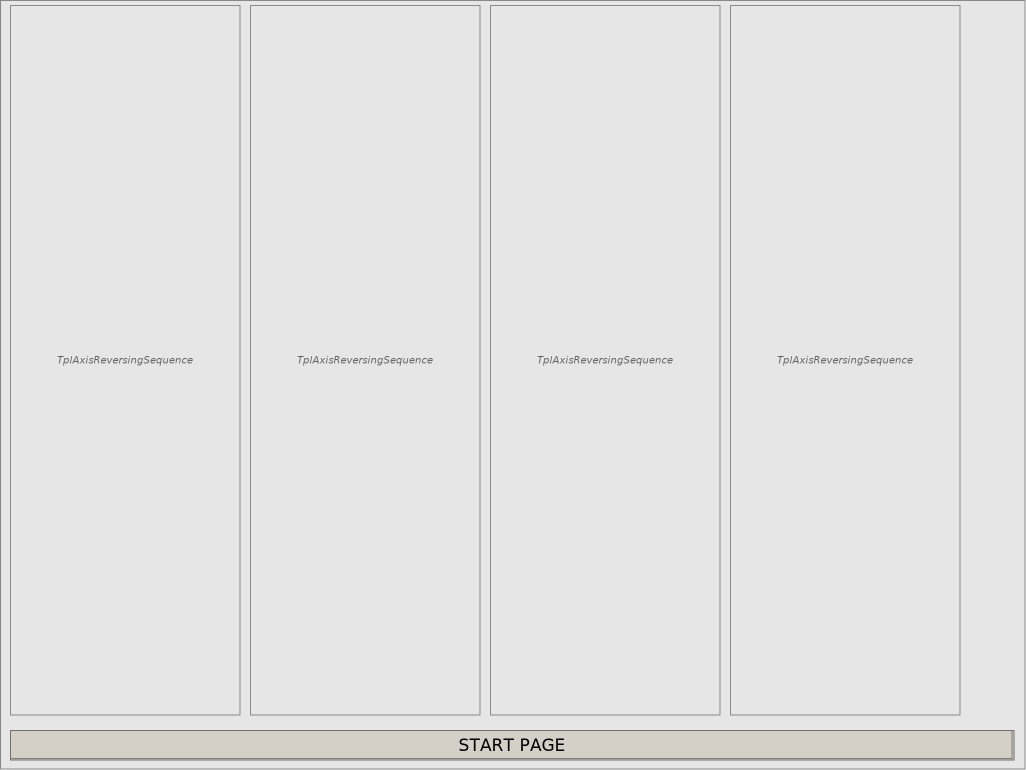
VISUALIZATION HmiAxisReversingSequence  // 1026x770
    Rectangle (0,0 1024x768)
    Button (10,730 1004x30), "START PAGE"
        OnMouseClick: change screen: HmiStartPage
    Frame (10,5 230x710)
        shows TplAxisReversingSequence(sAxisDescription := Axis1.sAxisDescription, fAbsolutePositon := stAxis1.NcToPlc.ActPos, fModuloPositon := stAxis1.NcToPlc.ModuloActPos, bError := Axis1.bAxisErr, nErrorId := Axis1.nAxisErrId, bReset := Axis1.bReset, bPowerStatus := Axis1.fbAxis.bPowerStatus, bReferenceCam := bStepperReferenceCam, bRevSeqStart := Axis1.bRevSeqStart, bRevSeqStop := Axis1.fbAxis.bRevSeqStop, fRevSeqTargetPos1 := Axis1.fbAxis.fRevSeqTargetPos1, fRevSeqTargetVelo1 := Axis1.fbAxis.fRevSeqTargetVelo1, fRevSeqTargetPos2 := Axis1.fbAxis.fRevSeqTargetPos2, fRevSeqTargetVelo2 := Axis1.fbAxis.fRevSeqTargetVelo2, nRevSeqIdleTime := Axis1.fbAxis.nRevSeqIdleTime, bRevSeqDone := Axis1.fbAxis.bRevSeqDone, bRevSeqBusy := Axis1.fbAxis.bRevSeqBusy)
    Frame (250,5 230x710)
        shows TplAxisReversingSequence(sAxisDescription := Axis2.sAxisDescription, fAbsolutePositon := stAxis2.NcToPlc.ActPos, fModuloPositon := stAxis2.NcToPlc.ModuloActPos, bError := Axis2.bAxisErr, nErrorId := Axis2.nAxisErrId, bReset := Axis2.bReset, bPowerStatus := Axis2.fbAxis.bPowerStatus, bReferenceCam := bAxis2ReferenceCamEL7, bRevSeqStart := Axis2.bRevSeqStart, bRevSeqStop := Axis2.fbAxis.bRevSeqStop, fRevSeqTargetPos1 := Axis2.fbAxis.fRevSeqTargetPos1, fRevSeqTargetVelo1 := Axis2.fbAxis.fRevSeqTargetVelo1, fRevSeqTargetPos2 := Axis2.fbAxis.fRevSeqTargetPos2, fRevSeqTargetVelo2 := Axis2.fbAxis.fRevSeqTargetVelo2, nRevSeqIdleTime := Axis2.fbAxis.nRevSeqIdleTime, bRevSeqDone := Axis2.fbAxis.bRevSeqDone, bRevSeqBusy := Axis2.fbAxis.bRevSeqBusy)
    Frame (490,5 230x710)
        shows TplAxisReversingSequence(sAxisDescription := Axis3.sAxisDescription, fAbsolutePositon := stAxis3.NcToPlc.ActPos, fModuloPositon := stAxis3.NcToPlc.ModuloActPos, bError := Axis3.bAxisErr, nErrorId := Axis3.nAxisErrId, bReset := Axis3.bReset, bPowerStatus := Axis3.fbAxis.bPowerStatus, bReferenceCam := AxisGeneral.bAxis3ReferenceCam, bRevSeqStart := Axis3.bRevSeqStart, bRevSeqStop := Axis3.fbAxis.bRevSeqStop, fRevSeqTargetPos1 := Axis3.fbAxis.fRevSeqTargetPos1, fRevSeqTargetVelo1 := Axis3.fbAxis.fRevSeqTargetVelo1, fRevSeqTargetPos2 := Axis3.fbAxis.fRevSeqTargetPos2, fRevSeqTargetVelo2 := Axis3.fbAxis.fRevSeqTargetVelo2, nRevSeqIdleTime := Axis3.fbAxis.nRevSeqIdleTime, bRevSeqDone := Axis3.fbAxis.bRevSeqDone, bRevSeqBusy := Axis3.fbAxis.bRevSeqBusy)
    Frame (730,5 230x710)
        shows TplAxisReversingSequence(sAxisDescription := Axis4.sAxisDescription, fAbsolutePositon := stAxis4.NcToPlc.ActPos, fModuloPositon := stAxis4.NcToPlc.ModuloActPos, bError := Axis4.bAxisErr, nErrorId := Axis4.nAxisErrId, bReset := Axis4.bReset, bPowerStatus := Axis4.fbAxis.bPowerStatus, bReferenceCam := AxisGeneral.bAxis4ReferenceCam, bRevSeqStart := Axis4.bRevSeqStart, bRevSeqStop := Axis4.fbAxis.bRevSeqStop, fRevSeqTargetPos1 := Axis4.fbAxis.fRevSeqTargetPos1, fRevSeqTargetVelo1 := Axis4.fbAxis.fRevSeqTargetVelo1, fRevSeqTargetPos2 := Axis4.fbAxis.fRevSeqTargetPos2, fRevSeqTargetVelo2 := Axis4.fbAxis.fRevSeqTargetVelo2, nRevSeqIdleTime := Axis4.fbAxis.nRevSeqIdleTime, bRevSeqDone := Axis4.fbAxis.bRevSeqDone, bRevSeqBusy := Axis4.fbAxis.bRevSeqBusy)
END_VISUALIZATION

(* stored: Version 1.1.0.1
   Visu HmiAxisReversingSequence: Id {4a2ed46e-f9f5-46f5-a439-d78a2e35232e} *)
